
FUNCTION CB_word_to_bool : BOOL


TITLE = ' Convert a word into a boolean '
VERSION : '1.0'
AUTHOR  : CB
NAME    : wordToBo
FAMILY  : TNI

VAR_INPUT
    IN : WORD;
END_VAR

BEGIN

CB_word_to_bool := (WORD_TO_INT(IN) <>0);

END_FUNCTION
